(* PLC project liner_cyclic.project, CODESYS CODESYS V3.5 SP17 Patch 3 *)
(* stored: creationDateTime 1970-01-01T00:00:00, modificationDateTime 1970-01-01T00:00:00 *)

FUNCTION_BLOCK Filter_AIO
  VAR_INPUT
    in : REAL;
    time_const : REAL;  (* постоянная времени фильтра 1000 = 1 сек *)
  END_VAR
  VAR_OUTPUT
    out : REAL;
  END_VAR

            IF time_const = 0 THEN
	out := in;
	ELSE
	out := (in - out) / time_const + out;		
	END_IF
          
END_FUNCTION_BLOCK
